# EPICS autosave request: support/dac128V-2-6/dac128VApp/Db/singleDAC_settings.req
#FILE... DAC_settings.req
#USAGE... DAC.db fields autosave'd.
$(P)DAC$(D)_$(N).DESC
$(P)DAC$(D)_$(N).VAL
$(P)DAC$(D)_$(N)_pulse.VAL
$(P)DAC$(D)_$(N)_tweakVal.VAL
